// Implicitly generated code : DO NOT EDIT
FUNCTION CheckLRangeSigned : LINT
VAR_INPUT
	value, lower, upper: LINT;
END_VAR

// Implicitly generated code : Only an Implementation suggestion
{noflow}
IF (value < lower) THEN
	CheckLRangeSigned := lower;
ELSIF(value > upper) THEN
	CheckLRangeSigned := upper;
ELSE
	CheckLRangeSigned := value;
END_IF

{flow}

END_FUNCTION

(* stored: Version 1.1.0.1, ProductVersion 3.1.4024.13
   POU CheckLRangeSigned: Id {2798c113-256f-4b0f-afd9-bd1deda5cdea}, SpecialFunc CheckLRangeSigned *)
